// Mitsubishi GX Works2 project: 21-05-2020 Control water level   PLC: FX3G

PROGRAM MAIN
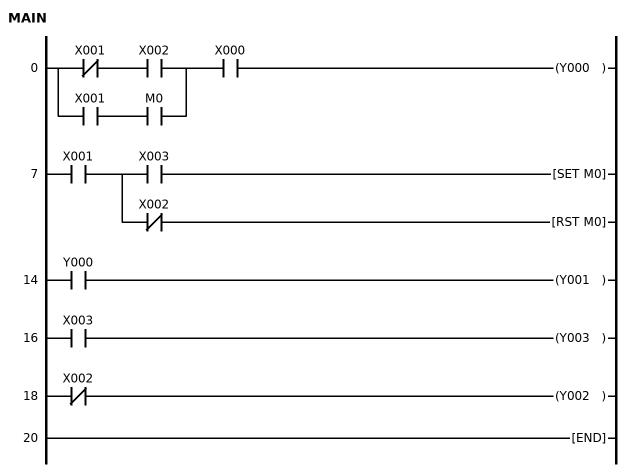
0     LDI     X001
      AND     X002
      LD      X001
      AND     M0
      ORB
      AND     X000
      OUT     Y000
7     LD      X001
      MPS
      AND     X003
      SET     M0
      MPP
      ANI     X002
      RST     M0
14    LD      Y000
      OUT     Y001
16    LD      X003
      OUT     Y003
18    LDI     X002
      OUT     Y002
20    END
END_PROGRAM
